PROGRAM MAIN
VAR

	bInit : BOOL := TRUE;	
	fbEvaluateOffsets: EvaluateAllOffsets; // Instance of EvaluateAllOffsets
END_VAR

(*
		This project reads the voltages from the Loadcell and transmits the data across ADS.
		
		1. Connect variables to hardware
		2. Read the voltage of each channel
		3. Convert from binary to float
		4. transmit across ADS

*)

// Initiliase the offsets and transmission variables
IF (bInit) THEN
	
	// Call the fucntion block that evaluates all the offsets
	fbEvaluateOffsets();
	
	GVL_Transmit.fTransmitAI1 := 0.0;
	GVL_Transmit.fTransmitAI2 := 0.0;
	GVL_Transmit.fTransmitAI3 := 0.0;
	GVL_Transmit.fTransmitAI4 := 0.0;
	GVL_Transmit.fTransmitAI5 := 0.0;
	GVL_Transmit.fTransmitAI6 := 0.0;
	
	bInit := FALSE;

END_IF

// Check whether to recalculate offsets
IF (GVL_Receive.bCalculateOffset) THEN
	// Call the fucntion block that evaluates all the offsets
	fbEvaluateOffsets();
	
	GVL_Receive.bCalculateOffset := FALSE;

END_IF

// If ready to recieve, scale and transmit the data
IF (GVL_Receive.bTransmitVoltages) THEN

	// Update the Globals which will be transmitted to the control PC
	GVL_Transmit.fTransmitAI1 := (ScaleVoltage(GVL_Receive.iRawAI1)) + GVL_Receive.fOffsetAI1;
	GVL_Transmit.fTransmitAI2 := (ScaleVoltage(GVL_Receive.iRawAI2)) + GVL_Receive.fOffsetAI2;
	GVL_Transmit.fTransmitAI3 := (ScaleVoltage(GVL_Receive.iRawAI3)) + GVL_Receive.fOffsetAI3;
	GVL_Transmit.fTransmitAI4 := (ScaleVoltage(GVL_Receive.iRawAI4)) + GVL_Receive.fOffsetAI4;
	GVL_Transmit.fTransmitAI5 := (ScaleVoltage(GVL_Receive.iRawAI5)) + GVL_Receive.fOffsetAI5;
	GVL_Transmit.fTransmitAI6 := (ScaleVoltage(GVL_Receive.iRawAI6)) + GVL_Receive.fOffsetAI6;
	
ELSE
	
	// Not ready to transmit, only write 0.0 to the Transmit GVLs
	GVL_Transmit.fTransmitAI1 := 0.0;
	GVL_Transmit.fTransmitAI2 := 0.0;
	GVL_Transmit.fTransmitAI3 := 0.0;
	GVL_Transmit.fTransmitAI4 := 0.0;
	GVL_Transmit.fTransmitAI5 := 0.0;
	GVL_Transmit.fTransmitAI6 := 0.0;
	
END_IF

END_PROGRAM

(* stored: Version 1.1.0.1, ProductVersion 3.1.4024.15
   POU MAIN: Id {4ef0117a-ae99-4538-91dd-8e8f23027317}, SpecialFunc None *)
